// TIA Portal V17 export
// export: Created 2023-02-14T02:49:37.1044754Z, ExportSetting WithDefaults, DisplayName Totally Integrated Automation Portal, DisplayVersion V17, DisplayName TIA Portal Openness, DisplayVersion V17, DisplayName TIA Portal Teamcenter Gateway, DisplayVersion V17, DisplayName TIA Portal Version Control Interface, DisplayVersion V17, DisplayName SINAMICS Startdrive Advanced, DisplayVersion V17, DisplayName SINAMICS Startdrive G130, G150, S120, S150, SINAMICS MV, S210, DisplayVersion V17, DisplayName SINAMICS Startdrive G110M, G120, G120C, G120D, G120P, G115D, DisplayVersion V17, DisplayName STEP 7 Professional, DisplayVersion V17, DisplayName STEP 7 Safety, DisplayVersion V17, DisplayName WinCC Professional, DisplayVersion V17
DATA_BLOCK "IO_Valve_T51_HW"   // DB311
VERSION : 0.1
// stored: AutoNumber false, DBAccessibleFromOPCUA true, DBAccessibleFromWebserver true, InstanceOfName IO Valve T51 HotWaterLine, InstanceOfType FB
"IO Valve T51 HotWaterLine"
   // VAR_INPUT
   //    lock : Bool;
   //    Init : Bool;
   //    testing : Bool;
   //    Reset : Bool;
   // END_VAR
   // VAR
   //    "AV-51.01" { S7_SetPoint := 'True'} : "Valve";
   //    "AV-51.02" { S7_SetPoint := 'True'} : "Valve";
   //    "AV-51.03" { S7_SetPoint := 'True'} : "Valve";
   //    "AV-51.04" { S7_SetPoint := 'True'} : "Valve";
   //    "AV-51.05" { S7_SetPoint := 'True'} : "Valve";
   //    "AV-51.06" { S7_SetPoint := 'True'} : "Valve";
   //    "AV-51.07" { S7_SetPoint := 'True'} : "Valve";
   //    "AV-51.08" { S7_SetPoint := 'True'} : "Valve";
   //    "AV-51.09" { S7_SetPoint := 'True'} : "Valve";
   //    "AV-51.10" { S7_SetPoint := 'True'} : "Valve";
   //    "AV-51.11" { S7_SetPoint := 'True'} : "Valve";
   //    "AV-51.12" { S7_SetPoint := 'True'} : "Valve";
   //    "AV-51.13" { S7_SetPoint := 'True'} : "Valve";
   //    "AV-51.14" { S7_SetPoint := 'True'} : "Valve";
   //    "AV-51.15" { S7_SetPoint := 'True'} : "Valve";
   //    "CV-51.11" { S7_SetPoint := 'True'} : "Valve";
   // END_VAR
BEGIN
END_DATA_BLOCK
